PROGRAM MAIN
VAR
	Machine : MachineModule := (Name := 'Machine');
END_VAR

Machine.CyclicLogic();

END_PROGRAM

(* stored: Version 1.1.0.1, ProductVersion 3.1.4024.12
   POU MAIN: Id {7bef8f53-b20c-4465-9e46-81406bba8435}, SpecialFunc None *)
